TEXTLIST TextList_Test_RP
  0 = 'tes trp' | FR: 'Test de remontée de pression' | EN: 'Pressure rise test'
  1 = 'init' | FR: 'Pression initiale' | EN: 'Initial pressure'
  2 = 'tps isol' | FR: "Durée d'isolement" | EN: 'Standby duration'
  3 = 'volume' | FR: 'Volume' | EN: 'Volume'
  4 = 'tps ecoul' | FR: 'Durée écoulée' | EN: 'Elapsed time'
  5 = 'result' | FR: 'Résultat :' | EN: 'Result:'
  6 = 'arret' | FR: 'Arrêt' | EN: 'Stop'
   = ''
END_TEXTLIST

(* stored: Version 1.1.0.1, ProductVersion 3.1.4024.10
   TextList TextList_Test_RP: Id {807aab10-fa02-44ce-8175-c92933fa0975} *)
